Staubli VAL3: WriteLine.pgx

public program WriteLine(num x_nFileID (dimensions=1), string x_sContext (dimensions=1), bool& x_bRes (dimensions=1))
  local num l_nNum
  local string l_sString
begin

  //文件标志符

  x_bRes=false
  if x_nFileID<0 or x_nFileID>9
    return
  endIf
  l_sString[0]=x_sContext
  //
  switch x_nFileID
    case 0
      l_nNum=$fileSet(0,l_sString,1)
    break

    case 1
      l_nNum=$fileSet(1,l_sString,1)
    break

    case 2
      l_nNum=$fileSet(2,l_sString,1)
    break

    case 3
      l_nNum=$fileSet(3,l_sString,1)
    break

    case 4
      l_nNum=$fileSet(4,l_sString,1)
    break

    case 5
      l_nNum=$fileSet(5,l_sString,1)
    break
    case 6
      l_nNum=$fileSet(6,l_sString,1)
    break

    case 7
      l_nNum=$fileSet(7,l_sString,1)
    break
    case 8
      l_nNum=$fileSet(8,l_sString,1)
    break

    case 9
      l_nNum=$fileSet(9,l_sString,1)
    break


  endSwitch
  if l_nNum!=1
    return
  endIf
  x_bRes=true


end
